Staubli VAL3: onBackEvent.pgx

program onBackEvent(bool& x_bSave[])
  local string l_sItem
  local num i
begin
//  //
//  // rename
//  //
//  call trajType:getTrajItem(l_tTraj,nIndex)
//  if l_tTraj.comment!=""
//    i=find(sEvent,l_tTraj.comment)
//  else
//    i=len(toString("",nIndex))+3
//  endIf
//  if i!=-1
//    // clean the line
//    call use:listcursor(use:nView,false)
//    // read the name
//    call use:read(40-use:nBottomX+i-1,nView+1,l_tTraj.comment,10,false)
//    call trajType:setTrajItem(l_tTraj,nIndex)
//    call buildList()
//    x_bSave=true
//  endIf
end
